PROGRAM PointerHelper

METHOD ReleaseDynamicMemory
VAR_INPUT
	value : POINTER TO BYTE;
	pointerType : POINTER_TYPE;
END_VAR
VAR
	objectPointer : POINTER TO Object;
END_VAR
IF value = 0 THEN
	RETURN;
END_IF

IF pointerType = POINTER_TYPE.OBJECT_POINTER THEN
	objectPointer := value;
	// to call FB_exit
	__DELETE(objectPointer);
ELSE
	__DELETE(value);
END_IF
END_METHOD

END_PROGRAM

(* stored: Version 1.1.0.1
   POU PointerHelper: Id {2efa693b-8ff2-4e0a-a84b-e316607e414f}, SpecialFunc None
   Method ReleaseDynamicMemory: Id {27594c08-0453-4d52-a64e-971260c6e1aa} *)
